# EPICS alarm handler configuration: mps_database/bareTest/alarms/areas/mpln_ltuh_mp02.alhConfig
GROUP NULL MPLN:LTUH:MP02:1
$ALIAS MPS Link Node 131
$GUIDANCE
LTUH MPS
   Group Name: MPLN:LTUH:MP02:1
   Summary PV:  MPLN:LTUH:MP02:1:STATSUMY
$END
CHANNEL  MPLN:LTUH:MP02:1    MPLN:LTUH:MP02:1:MPS_EN_RBV		-----
CHANNEL  MPLN:LTUH:MP02:1    MPLN:LTUH:MP02:1:LC1_MODE_RBV		-----
